Staubli VAL3: start.pgx

program start()
begin
  // This is the start program of the conveyor librairy
  call create(0)
  return
end
